// TIA Portal V15 export
// export: Created 2018-02-08T09:49:59.38156Z, ExportSetting None, DisplayName Totally Integrated Automation Portal, DisplayVersion V15, DisplayName TIA Portal Openness, DisplayVersion V15, DisplayName TIA Portal Teamcenter Gateway, DisplayVersion V15, DisplayName SINAMICS Startdrive Advanced, DisplayVersion V15, DisplayName G110M, G120, G120C, G120D, G120P, DisplayVersion V15, DisplayName G130, G150, S120, S150, SINAMICS MV, DisplayVersion V15, DisplayName STEP 7 Professional, DisplayVersion V15, DisplayName WinCC Professional, DisplayVersion V15, DisplayName SIMATIC Visualization Architect, DisplayVersion V15
FUNCTION "Workshop1_FC" : Void   // FC1, LAD
{ S7_Optimized_Access := 'TRUE' }
// stored: SetENOAutomatically False
   VAR_INPUT
      WaterLevel : Int;
      OilLevel : Int;
   END_VAR
BEGIN

REGION Network 1
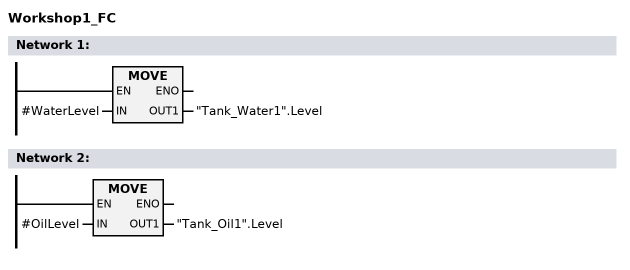
   RUNG wire#powerrail
      Move(in := #WaterLevel, out1 => "Tank_Water1".Level)
   END_RUNG
   // the same network as SCL:
   "Tank_Water1".Level := #WaterLevel;
END_REGION

REGION Network 2
   RUNG wire#powerrail
      Move(in := #OilLevel, out1 => "Tank_Oil1".Level)
   END_RUNG
   // the same network as SCL:
   "Tank_Oil1".Level := #OilLevel;
END_REGION
END_FUNCTION
